{attribute addProperty BoxType "EK1122-0000-0018"}
{attribute addProperty Id "Beckhoff_EPP6xxxsub_EK1100EK1100_179A0949162A_0001_EPP6001_0002_0016EPP6001_4599C92248060A_0002_EPP6001_0002_0017EPP6001_4599C92248060A_0003_EPP6001_0002_0018EPP6001_4599C92248060A_0004_EPP6002_0002_0016EPP6002_6961C256864108A_0005_EPP6002_0002_0017EPP6002_6961C256864108A_0006_EPP6002_0002_0018EPP6002_E45E7FFD864108A_0007_EPP6002_0002_0019EPP6002_E45E7FFD864108A_0008_EPP6090_0000_0017EPP6090_C46C03A814418A_0009_EPP6228_0022_0016EPP6228_8FEFBC8C28836"}
{attribute addProperty CRC "2966435658"}
{attribute addProperty SizeInBites "5344"}
{attribute addProperty SizeInBytes "668"}
TYPE Beckhoff_EPP6xxxEK1122_B0D0374A EXTENDS EK1122_179A0949 :
STRUCT
	{attribute addProperty Name "Beckhoff_EPP6xxxsub_EK1100"}
	Beckhoff_EPP6xxxsub_EK1100 : EK1100_179A0949;
	{attribute addProperty Name "A_0001_EPP6001_0002_0016"}
	A_0001_EPP6001_0002_0016 : EPP6001_4599C922;
	{attribute addProperty Name "A_0002_EPP6001_0002_0017"}
	A_0002_EPP6001_0002_0017 : EPP6001_4599C922;
	{attribute addProperty Name "A_0003_EPP6001_0002_0018"}
	A_0003_EPP6001_0002_0018 : EPP6001_4599C922;
	{attribute addProperty Name "A_0004_EPP6002_0002_0016"}
	A_0004_EPP6002_0002_0016 : EPP6002_6961C256;
	{attribute addProperty Name "A_0005_EPP6002_0002_0017"}
	A_0005_EPP6002_0002_0017 : EPP6002_6961C256;
	{attribute addProperty Name "A_0006_EPP6002_0002_0018"}
	A_0006_EPP6002_0002_0018 : EPP6002_E45E7FFD;
	{attribute addProperty Name "A_0007_EPP6002_0002_0019"}
	A_0007_EPP6002_0002_0019 : EPP6002_E45E7FFD;
	{attribute addProperty Name "A_0008_EPP6090_0000_0017"}
	A_0008_EPP6090_0000_0017 : EPP6090_C46C03A8;
	{attribute addProperty Name "A_0009_EPP6228_0022_0016"}
	A_0009_EPP6228_0022_0016 : EPP6228_8FEFBC8C;
END_STRUCT
END_TYPE

(* stored: Version 1.2.0.0, ProductVersion 3.1.4024.9
   DUT Beckhoff_EPP6xxxEK1122_B0D0374A: Id {86edca0f-b538-44d2-914e-887dc5034fdf} *)
